// TIA Portal project "ControleReservatorioAguaUdemyEX" (V14)
// Projeto de controle de reservatorio de agua, controle de nivel e acionamentos de motoresbombas

(* hardware
DEVICE "S71500/ET200MP station_1"  S7-1500 station
   slot 0: "Rail_0"  Rack  6ES7 590-1***0-0AA0
   slot 1: "PLC_1"  CPU 1511C-1 PN  6ES7 511-1CK00-0AB0  V2.1
      slot 3: "CPU display_1"  6ES7591-1AA00-0AA0
*)

// ===== PLC "PLC_1"  CPU 1511C-1 PN =====

VAR_GLOBAL   // PLC tag table "Default tag table"
   "Volume atual Tanque IO" AT %IW1 : Int;
   "Sensor Nivel Baixo IO" AT %I3.0 : Bool;
   "Sensor de Nivel Alto IO" AT %I2.0 : Bool;
   "Bomba B01 IO" AT %Q0.0 : Bool;
   "Alarme Nivel Baixo IO" AT %Q1.0 : Bool;
   "Alarme Nivel Alto IO" AT %Q2.0 : Bool;
END_VAR

DATA_BLOCK "EntradasINPUT"   // DB1
{ S7_Optimized_Access := 'TRUE' }
VERSION : 0.1
   VAR
      "Volume Total Tanque" : Real := 100.0;
      "Volume Atual Tanque" : Real;
      "Sensor de Nivel Baixo" : Bool;
      "Sensor de Nivel Alto" : Bool;
   END_VAR
BEGIN
END_DATA_BLOCK

DATA_BLOCK "SaidaOUTPUT"   // DB2
{ S7_Optimized_Access := 'TRUE' }
VERSION : 0.1
   VAR
      "Bomba B01" : Bool;
      "Alarme de Nivel Baixo" : Bool;
      "Alarme de Nivel Alto" : Bool;
   END_VAR
BEGIN
END_DATA_BLOCK

DATA_BLOCK "Controle e Registro do Reservatorio_DB"   // DB3
{ S7_Optimized_Access := 'TRUE' }
VERSION : 0.1
// stored: InstanceOfName Controle e Registro do Reservatorio
"Controle e Registro do Reservatorio"
BEGIN
   "Volume Total BLK" := 100.0;
END_DATA_BLOCK

FUNCTION_BLOCK "Controle e Registro do Reservatorio"   // FB1, LAD
{ S7_Optimized_Access := 'TRUE' }
VERSION : 0.1
   VAR_INPUT
      "Volume Total BLK" : Real;
      "Volume Atual BLK" : Real;
      "Sensor de nivel Baixo BLK" : Bool;
      "Sensor de Nivel Alto BLK" : Bool;
   END_VAR
   VAR_OUTPUT
      "Bomba BLK" : Bool;
      "Alarme Baixo BLK" : Bool;
      "Alarme Alto BLK" : Bool;
   END_VAR
   VAR
      "Registro Sensor Baixo BLK" : Array[0..100] of Date_And_Time;
      "IndexRegistro BLK" : Int;
      "AuxRegistro BLK" : Bool;
      "DateTime BLK" : Date_And_Time;
      "VolumeAtualPorcentagem BLK" : Real;
      "Ret_Val BLK" : Int;
   END_VAR
BEGIN

REGION Network 1: Sensor de nivel baixo
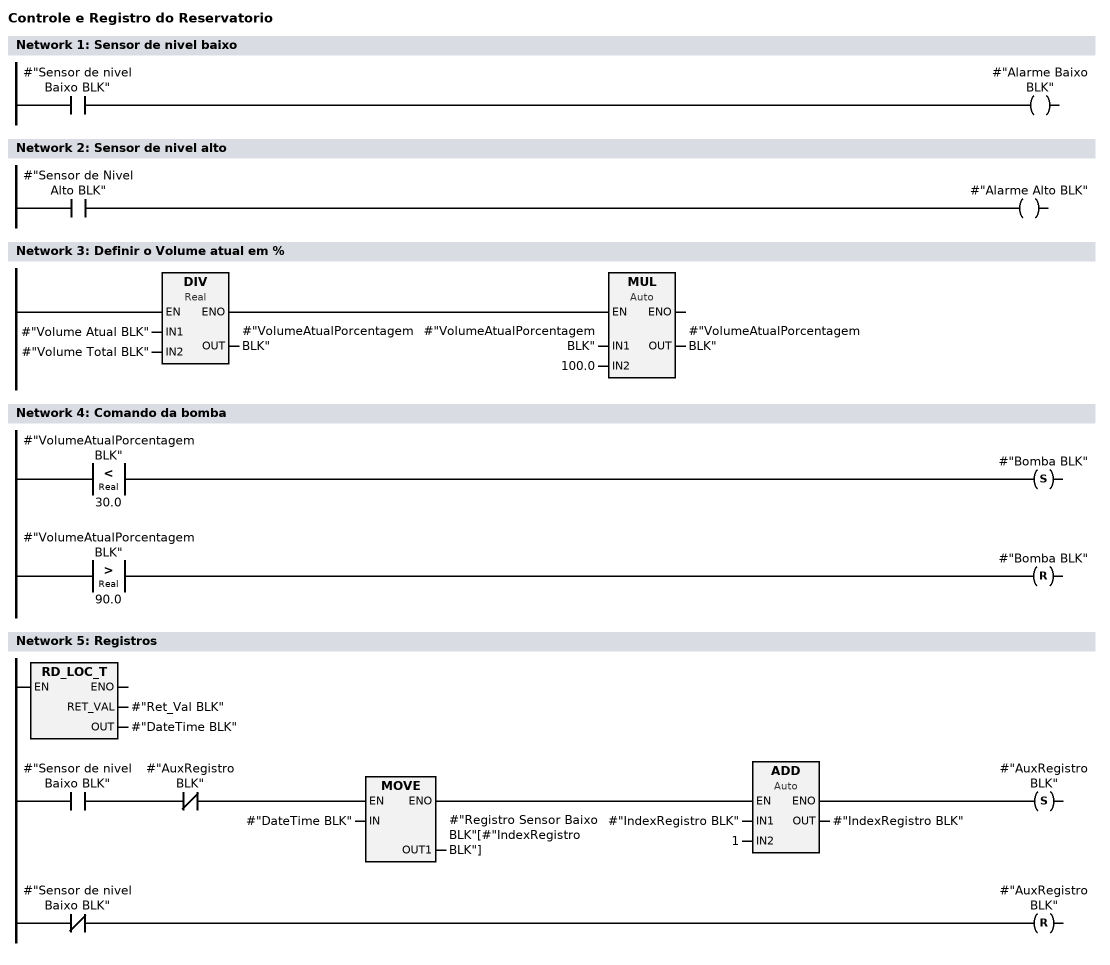
   RUNG wire#powerrail
      Contact( #"Sensor de nivel Baixo BLK" )
      Coil( #"Alarme Baixo BLK" )
   END_RUNG
   // the same network as SCL:
   #"Alarme Baixo BLK" := #"Sensor de nivel Baixo BLK";
END_REGION

REGION Network 2: Sensor de nivel alto
   RUNG wire#powerrail
      Contact( #"Sensor de Nivel Alto BLK" )
      Coil( #"Alarme Alto BLK" )
   END_RUNG
   // the same network as SCL:
   #"Alarme Alto BLK" := #"Sensor de Nivel Alto BLK";
END_REGION

REGION Network 3: Definir o Volume atual em %
   RUNG wire#powerrail
      { S7_Templates := "SrcType := Real" } Div(in1 := #"Volume Atual BLK", in2 := #"Volume Total BLK", out => #"VolumeAtualPorcentagem BLK")
      Mul(in1 := #"VolumeAtualPorcentagem BLK", in2 := 100.0, out => #"VolumeAtualPorcentagem BLK")
   END_RUNG
   // the same network as SCL:
   #"VolumeAtualPorcentagem BLK" := #"Volume Atual BLK" / #"Volume Total BLK";
   #"VolumeAtualPorcentagem BLK" := #"VolumeAtualPorcentagem BLK" * 100.0;
END_REGION

REGION Network 4: Comando da bomba
   RUNG wire#powerrail
      { S7_Templates := "SrcType := Real" } LT_Contact(in1 := #"VolumeAtualPorcentagem BLK", in2 := 30.0)
      S_Coil( #"Bomba BLK" )
   END_RUNG
   RUNG wire#powerrail
      { S7_Templates := "SrcType := Real" } GT_Contact(in1 := #"VolumeAtualPorcentagem BLK", in2 := 90.0)
      R_Coil( #"Bomba BLK" )
   END_RUNG
   // the same network as SCL:
   IF #"VolumeAtualPorcentagem BLK" < 30.0 THEN #"Bomba BLK" := TRUE; END_IF;
   IF #"VolumeAtualPorcentagem BLK" > 90.0 THEN #"Bomba BLK" := FALSE; END_IF;
END_REGION

REGION Network 5: Registros
   #"Ret_Val BLK" := RD_LOC_T(OUT => #"DateTime BLK");
   IF #"Sensor de nivel Baixo BLK" AND NOT #"AuxRegistro BLK" THEN
       #"Registro Sensor Baixo BLK"[#"IndexRegistro BLK"] := #"DateTime BLK";
       #"IndexRegistro BLK" := #"IndexRegistro BLK" + 1;
       #"AuxRegistro BLK" := TRUE;
   END_IF;
   IF NOT #"Sensor de nivel Baixo BLK" THEN #"AuxRegistro BLK" := FALSE; END_IF;
END_REGION
END_FUNCTION_BLOCK

FUNCTION "ConverDBtoIO" : Void   // FC1, SCL
{ S7_Optimized_Access := 'TRUE' }
VERSION : 0.1
BEGIN
   // Entradas DB para I/O CLP

   "EntradasINPUT"."Volume Atual Tanque" := "Volume atual Tanque IO";
   "EntradasINPUT"."Sensor de Nivel Baixo" := "Sensor Nivel Baixo IO";
   "EntradasINPUT"."Sensor de Nivel Alto" := "Sensor de Nivel Alto IO";

   //Saidas DB para I/O CLP
   "Bomba B01 IO":= "SaidaOUTPUT"."Bomba B01" ;
   "Alarme Nivel Alto IO":= "SaidaOUTPUT"."Alarme de Nivel Alto" ;
   "Alarme Nivel Baixo IO":= "SaidaOUTPUT"."Alarme de Nivel Baixo" ;
END_FUNCTION

ORGANIZATION_BLOCK "Main"   // OB1, LAD, ProgramCycle
TITLE = "Main Program Sweep (Cycle)"
{ S7_Optimized_Access := 'TRUE' }
VERSION : 0.1
   VAR_INPUT
      Initial_Call : Bool;   // Initial call of this OB
      Remanence : Bool;   // =True, if remanent data are available
   END_VAR
BEGIN

REGION Network 1
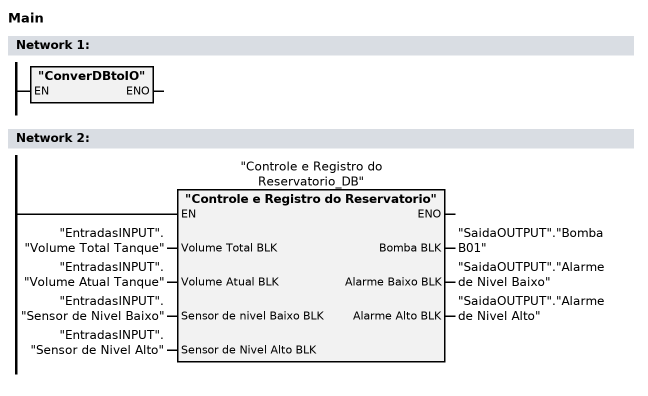
   RUNG wire#powerrail
      "ConverDBtoIO"()
   END_RUNG
   // the same network as SCL:
   "ConverDBtoIO"();
END_REGION

REGION Network 2
   RUNG wire#powerrail
      "Controle e Registro do Reservatorio_DB"("Volume Total BLK" := "EntradasINPUT"."Volume Total Tanque", "Volume Atual BLK" := "EntradasINPUT"."Volume Atual Tanque", "Sensor de nivel Baixo BLK" := "EntradasINPUT"."Sensor de Nivel Baixo", "Sensor de Nivel Alto BLK" := "EntradasINPUT"."Sensor de Nivel Alto", "Bomba BLK" => "SaidaOUTPUT"."Bomba B01", "Alarme Baixo BLK" => "SaidaOUTPUT"."Alarme de Nivel Baixo", "Alarme Alto BLK" => "SaidaOUTPUT"."Alarme de Nivel Alto")
   END_RUNG
   // the same network as SCL:
   "Controle e Registro do Reservatorio_DB"("Volume Total BLK" := "EntradasINPUT"."Volume Total Tanque",   // "Controle e Registro do Reservatorio"
                           "Volume Atual BLK" := "EntradasINPUT"."Volume Atual Tanque",
                           "Sensor de nivel Baixo BLK" := "EntradasINPUT"."Sensor de Nivel Baixo",
                           "Sensor de Nivel Alto BLK" := "EntradasINPUT"."Sensor de Nivel Alto",
                           "Bomba BLK" => "SaidaOUTPUT"."Bomba B01",
                           "Alarme Baixo BLK" => "SaidaOUTPUT"."Alarme de Nivel Baixo",
                           "Alarme Alto BLK" => "SaidaOUTPUT"."Alarme de Nivel Alto");
END_REGION
END_ORGANIZATION_BLOCK